FUNCTION_BLOCK FB_DS_Zustandscheck
VAR_IN_OUT
	Zustand			: ST_DS_Zustand;
END_VAR
VAR_INPUT
	Parameter		:ST_DS_Parameter;
END_VAR
VAR_OUTPUT
END_VAR
VAR
END_VAR

(*
	Warnung_Code
		0:	Allgemein Warnung Pufferspeicher
		2:	Grenztemperaturen unter- oder ueberschritten
*)

(* Interne Stoerungen / Warnungen *)
(* Warnung - Grenztemperaturen unter- oder ueberschritten *)
Zustand.Warnung_Code.2	:= Zustand.Druck > Parameter.Druck_Max OR Zustand.Druck < Parameter.Druck_Min;

(* Warnmeldung *)
IF Zustand.Warnung_Code > 0 THEN
	Zustand.Warnung := TRUE;
ELSE
	Zustand.Warnung := FALSE;
END_IF;

END_FUNCTION_BLOCK

(* stored: Version 1.1.0.1, ProductVersion 3.1.4024.9
   POU FB_DS_Zustandscheck: Id {636de036-5b5c-433c-b08e-e3299b1a2bf2}, SpecialFunc None *)
